// TIA Portal V18 export
// export: Created 2025-12-01T17:51:10.8926253Z, ExportSetting None, DisplayName Totally Integrated Automation Portal, DisplayVersion V18 Update 5, DisplayName TIA Portal Openness, DisplayVersion V18 Update 5, DisplayName TIA Portal Teamcenter Gateway, DisplayVersion V18, DisplayName TIA Portal Version Control Interface, DisplayVersion V18, DisplayName STEP 7 Professional, DisplayVersion V18 Update 5, DisplayName STEP 7 Safety, DisplayVersion V18, DisplayName WinCC Professional, DisplayVersion V18 Update 5
DATA_BLOCK "ModeDB"   // DB2203
{ S7_Optimized_Access := 'FALSE' }
// stored: AutoNumber false
   VAR
      Gen { S7_SetPoint := 'True'} : "ModeGenStruct";
   END_VAR
BEGIN
END_DATA_BLOCK
